SUBAPPLICATION AE2_ILOCK_T_FF_TO_BOOL_EVENT (* Ein Kettenglied eines wechselseitig verriegelten Toggle-Flip-Flops via AE2-Bidirektional-Adapter (SOCKET/PLUG-Kette), Ausgang als BOOL Q + Event EO. Generisch fuer beliebig viele Teilnehmer nutzbar, indem PLUG des einen an SOCKET des naechsten angeschlossen wird. Schwester-Baustein zu MyLib::sys::AE2_ILOCK_T_FF_TO_AX (dort Ausgang als AX-Adapter statt BOOL+Event). *)
  (* Standard: 61499-2 *)
  (* Version 1.0, 2026-09-09, Franz Höpfinger, Meisterschulen am Ostbahnhof, Ausgelagert aus Uebung_004b3c_sub zur Wiederverwendung fuer weitere verriegelte Toggle-Ketten. *)
  PACKAGE MyLib::sys;
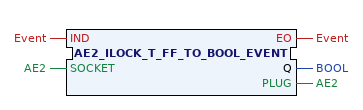
  EVENT_INPUT
    IND;
  END_EVENT
  EVENT_OUTPUT
    EO;
  END_EVENT
  VAR_OUTPUT
    Q : BOOL;
  END_VAR
  SOCKETS
    SOCKET : adapter::types::bidirectional::AE2;
  END_SOCKETS
  PLUGS
    PLUG : adapter::types::bidirectional::AE2;
  END_PLUGS
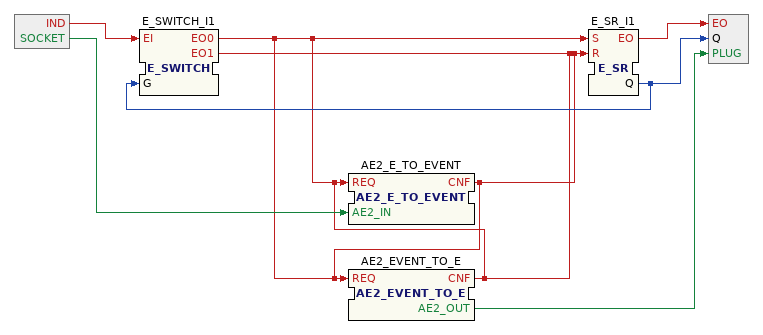
  FBS
    E_SR_I1 : iec61499::events::E_SR;
    E_SWITCH_I1 : iec61499::events::E_SWITCH;
    AE2_EVENT_TO_E : adapter::conversion::bidirectional::AE2_EVENT_TO_E;
    AE2_E_TO_EVENT : adapter::conversion::bidirectional::AE2_E_TO_EVENT;
  END_FBS
  EVENT_CONNECTIONS
    E_SWITCH_I1.EO0 TO E_SR_I1.S;
    E_SWITCH_I1.EO1 TO E_SR_I1.R;
    E_SR_I1.EO TO EO;
    IND TO E_SWITCH_I1.EI;
    E_SWITCH_I1.EO0 TO AE2_EVENT_TO_E.REQ;
    AE2_E_TO_EVENT.CNF TO E_SR_I1.R;
    AE2_EVENT_TO_E.CNF TO E_SR_I1.R;
    E_SWITCH_I1.EO0 TO AE2_E_TO_EVENT.REQ;
    AE2_E_TO_EVENT.CNF TO AE2_EVENT_TO_E.REQ;
    AE2_EVENT_TO_E.CNF TO AE2_E_TO_EVENT.REQ;
  END_CONNECTIONS
  DATA_CONNECTIONS
    E_SR_I1.Q TO E_SWITCH_I1.G;
    E_SR_I1.Q TO Q;
  END_CONNECTIONS
  ADAPTER_CONNECTIONS
    SOCKET TO AE2_E_TO_EVENT.AE2_IN;
    AE2_EVENT_TO_E.AE2_OUT TO PLUG;
  END_CONNECTIONS
END_SUBAPPLICATION
